(*
SPDX-FileCopyrightText: Â© 2026 Oleksandr Tiutyk <trofimich@gmail.com>
SPDX-License-Identifier: MIT
License: https://opensource.org/license/mit
*)

(*!
<summary>Exposes the task lifecycle and transition indicator for observation.</summary>
<description>
Borrows live backing variables supplied at initialization or rebound after online change. Getters safely guard
against unbound references and return default values if references are not valid. Treat the view and returned
references as read-only. Copy values when a snapshot is required.
</description>
*)

FUNCTION_BLOCK FINAL TaskState
VAR
	{attribute 'hide'} 
	_TaskState : REFERENCE TO TASK_STATE;
	{attribute 'hide'} 
	_TaskStateChanged : REFERENCE TO BOOL;
END_VAR

(*!
<summary>Binds the view to its owner's live state.</summary>
<description>
Stores references without copying their current values or changing the owner. Valid supplied references are
bound; skipped during online change copy code. Does not allocate or raise framework exceptions.
</description>
<param name="taskState">Live lifecycle state owned by the task.</param>
<param name="taskStateChanged">Live transition indicator owned by the task.</param>
*)
METHOD FB_Init: BOOL
VAR_INPUT
	bInitRetains : BOOL; // TRUE: the retain variables are initialized (reset warm / reset cold)
	bInCopyCode : BOOL;  // TRUE: the instance will be copied to the copy code afterward (online change)
	taskState : REFERENCE TO TASK_STATE;
	taskStateChanged : REFERENCE TO BOOL;
END_VAR
IF NOT bInCopyCode THEN
	Rebind(
		taskState := taskState,
		taskStateChanged := taskStateChanged
	);
END_IF
END_METHOD

(*!
<summary>Reports whether the task is READY.</summary>
<description>
READY permits Start; it does not imply a completed previous run. Returns FALSE if unbound.
</description>
*)
{attribute 'monitoring' := 'call'}
PROPERTY FINAL Ready : BOOL
GET
IF __ISVALIDREF(_TaskState) THEN
	Ready := _TaskState = TASK_STATE.READY;
END_IF
END_GET
END_PROPERTY

(*!
<summary>Rebinds the view to its owner's live state variables.</summary>
<description>
Updates internal references when valid variables are supplied. Used during initialization and
subsequent online-change reinitialization.
</description>
<param name="taskState">Live lifecycle state owned by the task.</param>
<param name="taskStateChanged">Live transition indicator owned by the task.</param>
*)
METHOD INTERNAL Rebind
VAR_INPUT
	taskState : REFERENCE TO TASK_STATE;
	taskStateChanged : REFERENCE TO BOOL;
END_VAR
IF __ISVALIDREF(taskState) THEN
	_TaskState REF= taskState;
END_IF

IF __ISVALIDREF(taskStateChanged) THEN
	_TaskStateChanged REF= taskStateChanged;
END_IF
END_METHOD

(*!
<summary>Reports whether the task is RUNNING.</summary>
<description>
Includes acquisition, processing, stopping and resource release. Returns FALSE if unbound.
</description>
*)
{attribute 'monitoring' := 'call'}
PROPERTY FINAL Running : BOOL
GET
IF __ISVALIDREF(_TaskState) THEN
	Running := _TaskState = TASK_STATE.RUNNING;
END_IF
END_GET
END_PROPERTY

(*!
<summary>Reports a lifecycle transition since the last Execute began.</summary>
<description>
Task.Execute clears this flag on entry, including when not running. Start, stopping and successful reset from
STOPPED can set it. It is not a count or a pulse tied to all PLC cycles. Returns FALSE if unbound.
</description>
*)
{attribute 'monitoring' := 'call'}
PROPERTY FINAL StateChanged : BOOL
GET
IF __ISVALIDREF(_TaskStateChanged) THEN
	StateChanged := _TaskStateChanged;
END_IF
END_GET
END_PROPERTY

(*!
<summary>Reports whether the task is STOPPED.</summary>
<description>
Read FinalStopReason for the result; stopping does not prove physical release. Returns FALSE if unbound.
</description>
*)
{attribute 'monitoring' := 'call'}
PROPERTY FINAL Stopped : BOOL
GET
IF __ISVALIDREF(_TaskState) THEN
	Stopped := _TaskState = TASK_STATE.STOPPED;
END_IF
END_GET
END_PROPERTY

(*!
<summary>Returns the current lifecycle state by value.</summary>
<description>
The returned enum is a snapshot of the borrowed backing state at this read. Returns READY if unbound.
</description>
*)
{attribute 'monitoring' := 'call'}
PROPERTY FINAL Value : TASK_STATE
GET
IF __ISVALIDREF(_TaskState) THEN
	Value := _TaskState;
END_IF
END_GET
END_PROPERTY

END_FUNCTION_BLOCK

(* stored: Version 1.1.0.1
   POU TaskState: Id {29e45909-ad82-4112-87e1-9792e16e3a41}, SpecialFunc None
   Folder Service methods: Id {c2ed99d1-9e97-4383-ae73-425083121bc7}
   Method FB_Init: Id {e5fa551c-3e84-40be-8ef7-9f3599da79cc}
   Property Ready: Id {752972e5-29e8-4d66-9b9b-bacbd95bc807}
   Get Get: Id {be7b15e3-99cc-422a-a1f5-1bf7586205fb}
   Method Rebind: Id {fa710b05-7cba-440f-9985-f97003992ddf}
   Property Running: Id {d518eb01-4363-42cc-ba1f-054fa911674c}
   Get Get: Id {ec791bbc-65ee-464b-aed3-27af2a7e3b0d}
   Property StateChanged: Id {600cdb42-d3b2-455a-b48f-83e96606c782}
   Get Get: Id {a6557db5-61fd-4ccb-85a4-b417b3791f73}
   Property Stopped: Id {3c595d3f-f42d-49d4-acc1-b271a058369a}
   Get Get: Id {746f2357-c572-4244-992a-04736fd48af0}
   Property Value: Id {aea1c285-89e6-43e8-af45-f9790e917087}
   Get Get: Id {41100485-bb0e-4be9-be0c-0ed2f158a278} *)
